FUNCTION_BLOCK FB_Lock
VAR_IN_OUT
	stInOut: ST_LockInOut;

END_VAR
VAR_INPUT
	bManualMode: BOOL;
	bReleaseOpening: BOOL;
END_VAR
VAR_OUTPUT
END_VAR
VAR
	bClosed: BOOL;
	bClosedAndLocked :BOOL;
	fbNotClosedTON:  TON;
	tNotClosed: TIME:=T#500MS;
	bReqOpen: BOOL;
	bReqManualOpen: BOOL;
	fbManualOpenTON: TON;
	tManualOpen: TIME:= T#10S;
	fbOpenningError:TON;
	tOpenningError: TIME:= T#3S;
	
END_VAR

bClosed := stInOut.bClosed;
bClosedAndLocked := stInOut.bClosed AND stInOut.bLocked;
fbNotClosedTON(IN:= NOT bClosed,PT:=tNotClosed);

fbManualOpenTON(IN:= bReqManualOpen,PT:=tManualOpen);
bReqManualOpen R=fbManualOpenTON.Q;

stInOut.bOpen:=(bReqOpen OR bReqManualOpen) AND bReleaseOpening;
fbOpenningError(IN:=stInOut.bOpen AND stInOut.bLocked, PT:=tOpenningError);   
bReqOpen := FALSE;

METHOD mManualOpen : BOOL
VAR_INPUT
END_VAR
IF bManualMode THEN
	bReqManualOpen := TRUE;
END_IF
END_METHOD

METHOD mOpen : BOOL
VAR_INPUT
END_VAR
IF NOT bManualMode THEN
	bReqOpen := TRUE;
END_IF
END_METHOD

{attribute 'monitoring':= 'call'}
PROPERTY prClosed : BOOL
GET
prClosed := bClosed;
END_GET
END_PROPERTY

{attribute 'monitoring':= 'call'}
PROPERTY prClosedAndLocked : BOOL
GET
prClosedAndLocked := bClosedAndLocked;
END_GET
END_PROPERTY

PROPERTY prNotClosed : BOOL
GET
prNotClosed := fbNotClosedTON.Q;
END_GET
END_PROPERTY

PROPERTY prOpeningError : BOOL
GET
prOpeningError := fbOpenningError.Q;
END_GET
END_PROPERTY

END_FUNCTION_BLOCK

(* stored: Version 1.1.0.1, ProductVersion 3.1.4024.15
   POU FB_Lock: Id {91f523f3-f163-4763-a4e6-4ed098eaffc8}, SpecialFunc None
   Method mManualOpen: Id {b8c17c3c-e745-4132-a0c7-08c3f6efe7a5}
   Method mOpen: Id {bc298bbe-e875-4372-832b-38d27168ff1a}
   Property prClosed: Id {2e6c38c2-a5e5-4f79-a46b-a0d10e0a3133}
   Get Get: Id {62c4d0ea-cbc1-4f11-9271-059fd6ea30b5}
   Property prClosedAndLocked: Id {add08f49-ff33-4490-b9a5-cdf9e877035a}
   Get Get: Id {e6280e40-c046-415f-8e5e-4b038e888555}
   Property prNotClosed: Id {c01d997c-215e-4190-8fc4-51334538e52b}
   Get Get: Id {d180bb63-f443-494a-9b61-999c19447b5f}
   Property prOpeningError: Id {bf9f24f8-5491-4903-970e-e6e6e04b48c3}
   Get Get: Id {2f921190-cea5-4dcf-8f1f-62ec53c880ca} *)
